(* CODESYS project Tc3_BAR_Common.library
   Company: Beckhoff
   Description: Library of implamentation common staff
   Version: 0.5.0
   DocFormat: reStructuredText
   Placeholder: Tc3_BAR_Common
   Author: Nikita Sakhnenko
   Title: Tc3_BAR_Common

Project tree, tasks and I/O mapping:
  libraries: Tc2_Standard, * (Beckhoff Automation GmbH); Tc2_System, * (Beckhoff Automation GmbH); Tc2_Utilities, * (Beckhoff Automation GmbH); VisuDialogs, * (System)
  Alarm/
    VisuElements/
      visualisation AlarmRecord_ActAlm_600
      visualisation AlarmRecord_History_600
      visualisation Current_Alarms_800x550
      visualisation Current_Alarms_dialog
      visualisation History_Of_Alarms_800x550
      visualisation History_Of_Alarms_dialog
    AlarmDiagram_1
    function block FB_Alarm [ST]: a1_Local_Quit, a2_Alarm_ScadaQuit, a3_Alarm_NoQuit, a4_Warning_RecordOnly, FB_init
    global variables LibAlarm
    program PRG_Alarms_Core [ST]: Blink, Current_Alarms_HMI, FB_Alarm_Execution, Get_Current_Time, History_Alarms_HMI
  Common/
    function TIME_TO_STRING_CE [ST]
    function TIME_TO_WSTRING_CE [ST]
    function TIME_TO_WSTRING_HMI [ST]
    function TS_to_STRING [ST]
    function TS_to_WSTRING [ST]
  DUTs/
    data type AlarmType
    data type E_AlarmColors
    data type ST_AlarmInfo
    data type ST_AlarmRecord
  InputVisu/
    visualisation TimeInput
  IO_terminals/
    DUTs/
      data type E_TermType
      data type TermChannel
    VisuElements/
      visualisation VisuAnalogChannel_Filled
      visualisation VisuAnalogChannel_Holow
    function block FB_AnalogChannel [ST]
  NC PTP Time Calculator/
    function block FB_7_SegTraj_Calculator [ST]: Step_1_Vmax_Amax_IsReachable, Step_2_Ta_Less_Than_Zero, Step_2_Td_Less_Than_Zero, Step_3_Gamma_Decrease_Seq
  Project Information/
    function F_GetCompany [ST]
    function F_GetTitle [ST]
    function F_GetVersion [ST]
  Trends/
    FBs/
      data type E_Trend_VISU_Type
      function block FB_TrendChanel [ST]: FB_init
      data type VisuStructPoint
    VISU/
      visualisation Trend_800_480
  Version/
    global variables Global_Version
  text list GlobalTextList
*)

// DUTs/AlarmType
{attribute 'qualified_only'}
{attribute 'strict'}
(*Вид аварийной блокировки*)
TYPE AlarmType :
(
	Alarm_LocalQuit 	:= 0,
	Alarm_ScadaQuit 	:= 1,
	Alarm_NoQuit 		:= 2,
	Warning_RecordOnly	:= 3,
	Warning_Type2		:= 4
);
END_TYPE

// DUTs/E_AlarmColors
{attribute 'qualified_only'}
{attribute 'strict'}
TYPE E_AlarmColors :
(
	E_Gray 		:= 16#7FD0D0D0, // Серый цвет
	E_Red  		:= 16#7FFF3C3C, // Красный цвет
	E_Yellow	:= 16#7FFFFF7D, // Желтый цвет
	E_green 	:= 16#7F00FF40, // Зеленый цвет
	E_Blue 		:= 16#7F8080FF  // Синий цвет
) DWORD;
END_TYPE

// DUTs/ST_AlarmInfo
(*Структура описания аварии*)
TYPE ST_AlarmInfo :
STRUCT
	AlarmID: WSTRING(5);				(*Текстовый идентификатор аварии*)
	Color: E_ALarmColors:=E_ALarmColors.E_Gray;		(*Цвет аварии. Заваисит от типа аварии*)
	Description: WSTRING(80):="--------------------------------------------------"; (*Поле описание аварии*)
	PossibleCause: WSTRING; 			(*Поле возможной причины аварии или указаний на аварийный узел*)
END_STRUCT
END_TYPE

// DUTs/ST_AlarmRecord
(*Структура записи в журнале аварий*)
TYPE ST_AlarmRecord EXTENDS ST_AlarmInfo :
STRUCT
	Time_On: 	WSTRING(20):="Нет данных"; 	(*Время возникновения аварии*)
	Time_Off: 	WSTRING(20):="Нет данных";	(*Время ухода аварии*)
	Time_Quit:	WSTRING(20):="Нет данных";	(*Время квитирования аварии*)
	isActive: BOOL;							(*Блокировка активна в настоящий момент*)
	wasQuited: BOOL;
END_STRUCT
END_TYPE

// IO_terminals/DUTs/E_TermType
{attribute 'qualified_only'}
{attribute 'strict'}
TYPE E_TermType :
(
	EL320x:=0,
	EL306x:=1,
	EL305x:=2,
	EL400x:=3,
	EL401x:=4,
	EL401x_4_20:=5
);
END_TYPE

// IO_terminals/DUTs/TermChannel
TYPE TermChannel :
STRUCT
	Status: WORD; (*бит XX.0 Underrange; бит ХХ.1 -Overrange; бит ХХ.6 - ERROR*)
	Value: INT;
END_STRUCT
END_TYPE

// Trends/FBs/E_Trend_VISU_Type
{attribute 'qualified_only'}
{attribute 'strict'}
TYPE E_Trend_VISU_Type :
(
	E_VISU_800_480 := 0,
	E_VISU_4_3 :=1
);
END_TYPE

// Trends/FBs/VisuStructPoint
TYPE VisuStructPoint :
STRUCT
	iX: INT;
	iY: INT;
END_STRUCT
END_TYPE

// Alarm/LibAlarm
{attribute 'qualified_only'}
VAR_GLOBAL CONSTANT
	MAX_ALARMS_NUM : UINT:=1000; (*Максимальное число аварий в программе*)
	MAX_HISTORY_NUM: UINT:=1000; (*Глубина Аварийного журнала*)
END_VAR

VAR_GLOBAL PERSISTENT
	HistoryAlarmsArray: ARRAY [1..MAX_ALARMS_NUM] OF ST_AlarmRecord; (*Массив с историей аварий*)
END_VAR

VAR_GLOBAL
	Blink: BOOL; // Мыргалка
	
	iNumberOfAlarms: UINT; 													//Количество экземпляров FB_Alarms
	FB_Alarm_Iterator: 	ARRAY [1..MAX_ALARMS_NUM] OF POINTER TO FB_alarm; 	//Итератор экземпляров FB_Alarm для исполнения
	ActiveAlarmsArray: 	ARRAY [1..MAX_ALARMS_NUM] OF ST_AlarmRecord; 		//Массив с текущими авариями
	
	Global_TimeStr: 		WSTRING(20);//	Метка текущего времени
	bRemoteQuitAllAlarms: 	BOOL;	 	// 	Переменная для удаленного квитирования аварии
	bLocalQuitAllAlarms AT %I*: BOOL;	//	Переменная для локального квитирования аварии
	bAlarmButtonBlink: 		BOOL;	 	// 	В настоящий момент есть активные не квитированные аварии требующие сброса
END_VAR

// Version/Global_Version
{attribute 'TcGenerated'}
{attribute 'no-analysis'}
{attribute 'linkalways'}
// This function has been automatically generated from the project information.
VAR_GLOBAL CONSTANT
	{attribute 'const_non_replaced'}
	stLibVersion_Tc3_BAR_Common : ST_LibVersion := (iMajor := 0, iMinor := 5, iBuild := 0, iRevision := 0, nFlags := 0, sVersion := '0.5.0');
END_VAR

// Alarm/FB_Alarm
{region "Documentation"}
(*
Функциональный блок обработки аварии
====================================
:Date: 2019-11-21
Служит для отображения аварий в текущем списке аварий и ведения истории.
В одном проекте может быть обьявлено максимум 1000 функциональных блоков FB_Alarm.
Максимальная глубина журнала аварий 1000.

Принцип использования
=====================
1. В библиотеке есть готовые экземпляры визуализации с таблицей текущих активных аварий: *Current_Alarms*
	и журналом аварий *History_Alarms*. Их следует добавить в проект, если есть необходимость в графическом отображении.
2. Перед обьявлением экземпляров обязательно следует добавить в исполняемый код программу *PRG_Alarms_Core();* 	 
	В этой подпрограмме происходят вызовы всех экземпляров FB_Alarm, а также всё необходимое для корректной работы системы вцелом.
3. После объявления *FB_Alarm*. Все что требуется для его использования это задать параметры и аварийное условие.

4. По переднему фронту *fbAlarm.AlarmEvent* активируется аварийная блокировка ("1" на выходе fbAlarm.isActive).
	 По заднему фронту входа *fbAlarm.AlarmEvent*Аварийная блокировкка снимется ("0" на выходе fbAlarm.isActive) в зависимости от типа аварии: 
====================  ========================================================
Alarm_Type           	Поведение по заднему фронту *fbAlarm.AlarmEvent*
====================  ========================================================
Local_Quit       		Снимается только после локального квитирования аварии
	 					LibAlarms.bLocalQuitAllAlarms - глобальная переменная 
						сброса квитирования всех активных аварий
						fbAlarm.bQuitAlarm - квитирование аварии экземпляра ФБ                 		
Alarm_ScadaQuit    		Снимается только после локального квитирования аварии
	 					LibAlarms.bLocalQuitAllAlarms - глобальная переменная 
						сброса квитирования всех активных аварий
	 					LibAlarms.bRemoteQuitAllAlarms - глобальная переменная 
						сброса квитирования всех активных аварий 							 
						fbAlarm.bQuitAlarm - квитирование аварии экземпляра ФБ
Alarm_NoQuit	    	Снимается сразу по заднему фронту *fbAlarm.AlarmEvent*
	 					Если не была квитирована, то об этом появиться запись в
						журнале
Warning_RecordOnly   	Делает запись в журнал по переднему фронту *fbAlarm.AlarmEvent*
    	 			 	Снимается без квитирования.
===================   ========================================================
5. Для отображения списка текущих аварий нужно использовать диалоговое окно TcSakhnenko.Current_Allarms_dialog
	 Для отображения журнала аварий нужно использовать диалоговое окно TcSakhnenko.History_Of_Allarms_dialog
*)
{endregion}
FUNCTION_BLOCK FINAL FB_Alarm	
VAR_INPUT
	AlarmCheckIsEnable: 		BOOL:=TRUE;		(*Проверка аварийного условия активна*)
	AlarmEvent: 				BOOL:=FALSE; 	(*Условие срабатывания аварии*)
	bQuitAlarm:    				BOOL:=FALSE;	(*Команда на квитирование аварии, 1-квитирование*)
	AlarmType: 					AlarmType; 		(*Тип квитирования аварии*)
	AlarmInfo: ST_AlarmInfo; 
	AlarmActivationDelay: 		TIME; 			(*Задержка на срабатывание аварии*)
END_VAR
VAR_OUTPUT
	isActive: BOOL; 		(*Аварийая блокировка активна*)
	WasQuited: BOOL;		(*Авария была квитирована*)
END_VAR
VAR
	tDelay : TON;
	TempAlarmRec: ST_AlarmRecord;
	AlarmNum: UINT; 			(*Порядковый номер аварии*)
	iState: UINT;(*Состояние аварии*)
	i: UINT;
	n: UINT;
END_VAR

IF AlarmCheckIsEnable THEN 
	CASE  AlarmType OF
		00:
			a1_Local_Quit();
		01:
			a2_Alarm_ScadaQuit();
		02:
			a3_Alarm_NoQuit();
		03:
			a4_Warning_RecordOnly();
	END_CASE
END_IF

ACTION a1_Local_Quit:
(*Обработчик Аварии, которую необходимо квитировать. Только локально.*)
TempAlarmRec.wasQuited:=WasQuited;
TempAlarmRec.isActive:=isActive;

CASE iState OF
	0:(*Инициализация*)
		isActive:=FALSE;
		WasQuited:=FALSE;
		TempAlarmRec.wasQuited:=FALSE;
		TempAlarmRec.Time_Quit:="Не квитирована";
		TempAlarmRec.AlarmID:=AlarmInfo.AlarmID;
		TempAlarmRec.Color:=AlarmInfo.Color;
		TempAlarmRec.Description:=AlarmInfo.Description;
		TempAlarmRec.PossibleCause:=AlarmInfo.PossibleCause;
 		iState:=10;

	10:(*Авария не активна. Ожидание активации аварии*)
		tDelay(IN:=AlarmEvent, PT:=AlarmActivationDelay);
			
		IF tDelay.Q THEN (*Возникновение первой аварии*)
			TempAlarmRec.PossibleCause:=AlarmInfo.PossibleCause;
			tDelay(IN:=FALSE);
			iState:=20;
		END_IF

		IF isActive THEN (*Авария не была квитирована и возникла еще раз*)
			TempAlarmRec.PossibleCause:=AlarmInfo.PossibleCause;
			tDelay(IN:=FALSE);
			iState:=30;
		END_IF
		
	20: (*Запись Времени Аварии*)
		TempAlarmRec.Time_On:=LibAlarm.Global_TimeStr;
		isActive:=TRUE;
		iState:= 30;
		
	30: (*Ожидание квитирования аварии и ее ухода*)
		IF (LibAlarm.bLocalQuitAllAlarms OR bQuitAlarm) THEN 
			TempAlarmRec.Time_Quit:=LibAlarm.Global_TimeStr;
			WasQuited:=TRUE;
			iState:=40;
		END_IF

		IF NOT AlarmEvent THEN
			IF NOT WasQuited THEN
				TempAlarmRec.Time_OFF:=LibAlarm.Global_TimeStr;
				iState:=31;
			END_IF;
		END_IF
	31:(*Авария ушла но не квитирована*)
			IF (LibAlarm.bLocalQuitAllAlarms OR bQuitAlarm) THEN
				TempAlarmRec.Time_Quit:=LibAlarm.Global_TimeStr;
				WasQuited:=TRUE;

				FOR i:=0 TO (LibAlarm.MAX_HISTORY_NUM - 2) DO
					n:=LibAlarm.MAX_HISTORY_NUM-i;
					LibAlarm.HistoryAlarmsArray[n]:=LibAlarm.HistoryAlarmsArray[n-1];
				END_FOR;

				LibAlarm.HistoryAlarmsArray[1]:=TempAlarmRec;
				iState:=00;
			END_IF
		
		IF AlarmEvent THEN //авария пришла снова
			TempAlarmRec.Time_Quit:="Не квитирована";

			FOR i:=0 TO (LibAlarm.MAX_HISTORY_NUM - 2) DO
				n:=LibAlarm.MAX_HISTORY_NUM-i;
				LibAlarm.HistoryAlarmsArray[n]:=LibAlarm.HistoryAlarmsArray[n-1];
			END_FOR;
		
			LibAlarm.HistoryAlarmsArray[1]:=TempAlarmRec;
			
			iState:=10;
		END_IF
		
		40:(*Авария ушла и квитирована*)
			IF NOT AlarmEvent THEN
			TempAlarmRec.Time_OFF:=LibAlarm.Global_TimeStr;

				FOR i:=0 TO (LibAlarm.MAX_HISTORY_NUM - 2) DO
					n:=LibAlarm.MAX_HISTORY_NUM-i;
					LibAlarm.HistoryAlarmsArray[n]:=LibAlarm.HistoryAlarmsArray[n-1];
				END_FOR;
		
				LibAlarm.HistoryAlarmsArray[1]:=TempAlarmRec;

				iState:=0;
			END_IF
		
END_CASE
END_ACTION

ACTION a2_Alarm_ScadaQuit:
(*Обработчик Аварии, которую необходимо квитировать. Локально и удаленно.*)
TempAlarmRec.wasQuited:=WasQuited;
TempAlarmRec.isActive:=isActive;

CASE iState OF
	0:(*Инициализация*)
		isActive:=FALSE;
		WasQuited:=FALSE;
		TempAlarmRec.Time_Quit:="Не квитирована";
		TempAlarmRec.AlarmID:=AlarmInfo.AlarmID;
		TempAlarmRec.Color:=AlarmInfo.Color;
		TempAlarmRec.Description:=AlarmInfo.Description;
		TempAlarmRec.PossibleCause:=AlarmInfo.PossibleCause;
 		iState:=10;

	10:(*Авария не активна. Ожидание активации аварии*)
		tDelay(IN:=AlarmEvent, PT:=AlarmActivationDelay);
			
		IF tDelay.Q THEN (*Возникновение первой аварии*)
			TempAlarmRec.PossibleCause:=AlarmInfo.PossibleCause;
			tDelay(IN:=FALSE);
			iState:=20;
		END_IF

		IF isActive THEN (*Авария не была квитирована и возникла еще раз*)
			TempAlarmRec.PossibleCause:=AlarmInfo.PossibleCause;
			tDelay(IN:=FALSE);
			iState:=30;
		END_IF
		
	20: (*Запись Времени Аварии*)
		TempAlarmRec.Time_On:=LibAlarm.Global_TimeStr;
		isActive:=TRUE;
		iState:= 30;
		
	30: (*Ожидание квитирования аварии и ее ухода*)
		IF (LibAlarm.bLocalQuitAllAlarms OR bQuitAlarm OR LibAlarm.bRemoteQuitAllAlarms) THEN 
			TempAlarmRec.Time_Quit:=LibAlarm.Global_TimeStr;
			WasQuited:=TRUE;
			iState:=40;
		END_IF

		IF NOT AlarmEvent THEN
			IF NOT WasQuited THEN
				TempAlarmRec.Time_OFF:=LibAlarm.Global_TimeStr;
				iState:=31;
			END_IF;
		END_IF
	31:(*Авария ушла но не квитирована*)
			IF (LibAlarm.bLocalQuitAllAlarms OR bQuitAlarm OR LibAlarm.bRemoteQuitAllAlarms) THEN
				TempAlarmRec.Time_Quit:=LibAlarm.Global_TimeStr;
				WasQuited:=TRUE;

				FOR i:=0 TO (LibAlarm.MAX_HISTORY_NUM - 2) DO
					n:=LibAlarm.MAX_HISTORY_NUM-i;
					LibAlarm.HistoryAlarmsArray[n]:=LibAlarm.HistoryAlarmsArray[n-1];
				END_FOR;

				LibAlarm.HistoryAlarmsArray[1]:=TempAlarmRec;
				iState:=00;
			END_IF

		IF AlarmEvent THEN
			TempAlarmRec.Time_Quit:="Не квитирована";

			FOR i:=0 TO (LibAlarm.MAX_HISTORY_NUM - 2) DO
				n:=LibAlarm.MAX_HISTORY_NUM-i;
				LibAlarm.HistoryAlarmsArray[n]:=LibAlarm.HistoryAlarmsArray[n-1];
			END_FOR;
		
			LibAlarm.HistoryAlarmsArray[1]:=TempAlarmRec;
			
			iState:=10;
		END_IF
		
		40:(*Авария ушла и квитирована*)
			IF NOT AlarmEvent THEN
			TempAlarmRec.Time_OFF:=LibAlarm.Global_TimeStr;

				FOR i:=0 TO (LibAlarm.MAX_HISTORY_NUM - 2) DO
					n:=LibAlarm.MAX_HISTORY_NUM-i;
					LibAlarm.HistoryAlarmsArray[n]:=LibAlarm.HistoryAlarmsArray[n-1];
				END_FOR;
		
				LibAlarm.HistoryAlarmsArray[1]:=TempAlarmRec;

				iState:=0;
			END_IF
		
END_CASE
END_ACTION

ACTION a3_Alarm_NoQuit:
(*Обработчик Аварии, которую необходимо квитировать*)
TempAlarmRec.wasQuited:=WasQuited;
TempAlarmRec.isActive:=isActive;

CASE iState OF
	0:(*Инициализация*)
		isActive:=FALSE;
		WasQuited:=FALSE;
		TempAlarmRec.Time_Quit:="Не квитирована";
		TempAlarmRec.AlarmID:=AlarmInfo.AlarmID;
		TempAlarmRec.Color:=AlarmInfo.Color;
		TempAlarmRec.Description:=AlarmInfo.Description;
		TempAlarmRec.PossibleCause:=AlarmInfo.PossibleCause;
 		iState:=10;

	10:(*Авария не активна. Ожидание активации аварии*)
		tDelay(IN:=AlarmEvent, PT:=AlarmActivationDelay);
			
		IF tDelay.Q THEN (*Возникновение первой аварии*)
			TempAlarmRec.PossibleCause:=AlarmInfo.PossibleCause;
			tDelay(IN:=FALSE);
			iState:=20;
		END_IF

		IF isActive THEN (*Авария не была квитирована и возникла еще раз*)
			TempAlarmRec.PossibleCause:=AlarmInfo.PossibleCause;
			tDelay(IN:=FALSE);
			iState:=30;
		END_IF
		
	20: (*Запись Времени Аварии*)
		TempAlarmRec.Time_On:=LibAlarm.Global_TimeStr;
		isActive:=TRUE;
		iState:= 30;
		
	30: (*Ожидание квитирования аварии и ее ухода*)
		IF (LibAlarm.bLocalQuitAllAlarms OR bQuitAlarm OR LibAlarm.bRemoteQuitAllAlarms) THEN 
			TempAlarmRec.Time_Quit:=LibAlarm.Global_TimeStr;
			WasQuited:=TRUE;
			iState:=40;
		END_IF

		IF NOT AlarmEvent THEN
			IF NOT WasQuited THEN
				TempAlarmRec.Time_OFF:=LibAlarm.Global_TimeStr;
				iState:=40;
			END_IF;
		END_IF
		
		40:(*Авария ушла и квитирована*)
			IF NOT AlarmEvent THEN
			TempAlarmRec.Time_OFF:=LibAlarm.Global_TimeStr;

				FOR i:=0 TO (LibAlarm.MAX_HISTORY_NUM - 2) DO
					n:=LibAlarm.MAX_HISTORY_NUM-i;
					LibAlarm.HistoryAlarmsArray[n]:=LibAlarm.HistoryAlarmsArray[n-1];
				END_FOR;
		
				LibAlarm.HistoryAlarmsArray[1]:=TempAlarmRec;

				iState:=0;
			END_IF
		
END_CASE
END_ACTION

ACTION a4_Warning_RecordOnly:
(*Предупреждение*)
CASE iState OF
	0:(*Инициализация*)
		isActive:=FALSE;
		WasQuited:=FALSE;
		TempAlarmRec.Time_Quit:="Не квитирована";
		TempAlarmRec.AlarmID:=AlarmInfo.AlarmID;
		TempAlarmRec.Color:=AlarmInfo.Color;
		TempAlarmRec.Description:=AlarmInfo.Description;
		TempAlarmRec.PossibleCause:=AlarmInfo.PossibleCause;
 		iState:=10;

	10:(*Авария не активна. Ожидание активации аварии*)
		tDelay(IN:=AlarmEvent, PT:=AlarmActivationDelay);
			
		IF tDelay.Q THEN (*Возникновение первой аварии*)
			tDelay(IN:=FALSE);
			
			TempAlarmRec.Time_ON:=LibAlarm.Global_TimeStr;
			TempAlarmRec.Time_Quit:="Не квитирована";
			TempAlarmRec.Time_OFF:=LibAlarm.Global_TimeStr;
			
				FOR i:=0 TO (LibAlarm.MAX_HISTORY_NUM - 2) DO
					n:=LibAlarm.MAX_HISTORY_NUM-i;
					LibAlarm.HistoryAlarmsArray[n]:=LibAlarm.HistoryAlarmsArray[n-1];
				END_FOR;
		
				LibAlarm.HistoryAlarmsArray[1]:=TempAlarmRec;
				
			iState:=20;
		END_IF

		
	20: (*Запись Времени Аварии*)
		IF NOT AlarmEvent THEN
			iState:=00;
		END_IF
		
END_CASE
END_ACTION

METHOD FB_init : BOOL
VAR_INPUT
	bInitRetains : BOOL; // if TRUE, the retain variables are initialized (warm start / cold start)
	bInCopyCode : BOOL;  // if TRUE, the instance afterwards gets moved into the copy code (online change)
END_VAR
libAlarm.iNumberOfAlarms:=libAlarm.iNumberOfAlarms+1;
AlarmNum:=libAlarm.iNumberOfAlarms;
LibAlarm.FB_Alarm_Iterator[AlarmNum]:=THIS;
END_METHOD

END_FUNCTION_BLOCK

// Alarm/PRG_Alarms_Core
PROGRAM PRG_Alarms_Core
VAR CONSTANT
	CurrentAlarmsDisplayNum: UINT:=10;//Количество отображаемых на экране текущих аварий
	HistoryAlarmsDisplayNum: UINT:=10;//Количество отображаемых на экране текущих аварий
END_VAR
VAR
	iFB: UINT; (*Итератор Функциональных блоков*)
	iCA: UINT; (*Итератор текущих аварий*)
	{region "Current_Alarms_HMI"}
	HMI_ActiveAlarms: ARRAY [1..CurrentAlarmsDisplayNum] OF ST_AlarmRecord;(*Масив с текущими отображаемыми авариями*)
	HMI_NumsAA : ARRAY[1..CurrentAlarmsDisplayNum] OF UINT;	(*Индексы в массиве текущих аварий*)
	iActiveAlarmsNumber: UINT;
	HMI_CurListAA: UINT;
	HMI_CurShiftAA: UINT;
	iHMI_AA: UINT;
	{endregion}
	
	{region "History_Alarms_HMI"}
	HMI_HistoryAlarms: ARRAY [1..HistoryAlarmsDisplayNum] OF ST_AlarmRecord;(*Масив с *)
	HMI_NumsHY : ARRAY[1..HistoryAlarmsDisplayNum] OF UINT;	(*Индексы в массиве истории аварий*)
	HMI_CurListHY: UINT;
	HMI_CurShiftHY: UINT;
	iHMI_HY: UINT;
	{endregion}
		 
	DefaultRec: ST_AlarmRecord;
	{region "Мыргалка"}
	t1: TON:=(PT:=T#1S);
	{endregion}
	
	{region "Get_Current_Time"}
	//Обновление строки текущего времени
	NT_GetTime: NT_GetTime;
	tonGetTime: TON:=(PT:=T#500MS);
	{endregion}
END_VAR

Get_Current_Time();

Blink();

FB_Alarm_Execution();

Current_Alarms_HMI();

History_Alarms_HMI();

ACTION Blink:
t1(in:=NOT t1.q);

IF t1.q THEN
LibAlarm.Blink:=NOT LibAlarm.Blink;
END_IF
END_ACTION

ACTION Current_Alarms_HMI:
	IF (HMI_CurShiftAA > LibAlarm.iNumberOfAlarms) THEN
		HMI_CurShiftAA:=LibAlarm.iNumberOfAlarms;
	ELSIF (HMI_CurShiftAA < 0 ) THEN
		HMI_CurShiftAA:=0;
	END_IF
	
	HMI_CurListAA := HMI_CurShiftAA / CurrentAlarmsDisplayNum;
	
	FOR iHMI_AA:=1 TO CurrentAlarmsDisplayNum DO
		HMI_NumsAA[iHMI_AA]:=iHMI_AA+HMI_CurShiftAA;
		HMI_ActiveAlarms[iHMI_AA]:=LibAlarm.ActiveAlarmsArray[HMI_NumsAA[iHMI_AA]];
	END_FOR
END_ACTION

ACTION FB_Alarm_Execution:
iCA:=1;
FOR iFB:=1 TO LibAlarm.iNumberOfAlarms DO
		LibAlarm.FB_Alarm_Iterator[iFB]^();
		LibAlarm.ActiveAlarmsArray[iFB]:=DefaultRec;
		IF LibAlarm.FB_Alarm_Iterator[iFB]^.isActive THEN
			LibAlarm.ActiveAlarmsArray[iCA]:=LibAlarm.FB_Alarm_Iterator[iFB]^.TempAlarmRec;
			iCA:=iCA+1;
		END_IF
END_FOR
END_ACTION

ACTION Get_Current_Time:
(*Получение текущего времени*)
tonGetTime(IN:= NOT tonGetTime.Q);
NT_GetTime(START:=tonGetTime.Q );
IF tonGetTime.Q THEN
	LibAlarm.Global_TimeStr := TS_to_WSTRING(NT_GetTime.TIMESTR);
END_IF
END_ACTION

ACTION History_Alarms_HMI:
	IF (HMI_CurShiftHY > (LibAlarm.MAX_HISTORY_NUM - HistoryAlarmsDisplayNum)) THEN
		HMI_CurShiftHY:=LibAlarm.MAX_HISTORY_NUM - HistoryAlarmsDisplayNum;
	ELSIF (HMI_CurShiftHY < 0 ) THEN
		HMI_CurShiftHY:=0;
	END_IF
	
	HMI_CurListHY := HMI_CurShiftHY / HistoryAlarmsDisplayNum;
	
	FOR iHMI_HY:=1 TO HistoryAlarmsDisplayNum DO
		HMI_NumsHY[iHMI_HY]:=iHMI_HY+HMI_CurShiftHY;
		HMI_HistoryAlarms[iHMI_HY]:=LibAlarm.HistoryAlarmsArray[HMI_NumsHY[iHMI_HY]];
	END_FOR
END_ACTION

END_PROGRAM

// Common/TS_to_WSTRING
FUNCTION TS_to_WSTRING : WSTRING(20)
VAR_INPUT
	in:TIMESTRUCT;
END_VAR
VAR
	str: WSTRING;
END_VAR

IF in.wHour>=10 THEN
str:=WCONCAT (str, WORD_TO_WSTRING(in.wHour));
ELSE
str:=WCONCAT (str, "0");
str:=WCONCAT (str, WORD_TO_WSTRING(in.wHour));
END_IF

str:=WCONCAT (str, ":");

IF in.wMinute>=10 THEN
str:=WCONCAT (str, WORD_TO_WSTRING(in.wMinute));
ELSE
str:=WCONCAT (str, "0");
str:=WCONCAT (str, WORD_TO_WSTRING(in.wMinute));
END_IF

str:=WCONCAT (str, ":");

IF in.wSecond>=10 THEN
str:=WCONCAT (str, WORD_TO_WSTRING(in.wSecond));
ELSE
str:=WCONCAT (str, "0");
str:=WCONCAT (str, WORD_TO_WSTRING(in.wSecond));
END_IF

str:=WCONCAT (str, " ");
str:=WCONCAT (str, WORD_TO_WSTRING(in.wDay));

IF in.wMonth <10 THEN
	str:=WCONCAT (str, ".0");
	str:=WCONCAT (str, WORD_TO_WSTRING(in.wMonth));	
ELSE
	str:=WCONCAT (str, ".");
	str:=WCONCAT (str, WORD_TO_WSTRING(in.wMonth));
END_IF

str:=WCONCAT (str, ".");
str:=WCONCAT (str, WORD_TO_WSTRING(in.wYear-2000));
TS_to_WSTRING:=str;

END_FUNCTION

// Common/TIME_TO_STRING_CE
FUNCTION TIME_TO_STRING_CE  : STRING(15)
VAR_INPUT
	InTime : TIME;
END_VAR
VAR
	DD: UINT;
	HH: UINT;
	MM: UINT;
	SS:UINT;
END_VAR

dd:=DWORD_TO_UINT (TIME_TO_DWORD(InTime) / TIME_TO_DWORD(T#1D));
HH:=DWORD_TO_UINT (TIME_TO_DWORD((InTime - T#24h*DD) / TIME_TO_DWORD(T#1h)));
MM:=DWORD_TO_UINT (TIME_TO_DWORD(InTime-T#24h*DD - T#60m*HH) / TIME_TO_DWORD(T#1m));
SS:=DWORD_TO_UINT (TIME_TO_DWORD(InTime - T#24h*DD - T#60m*HH - T#60s*MM) / TIME_TO_DWORD(T#1s));
TIME_TO_STRING_CE:=CONCAT(TIME_TO_STRING_CE, UINT_TO_STRING(DD));
TIME_TO_STRING_CE:=CONCAT(TIME_TO_STRING_CE, 'дн. ');
IF HH < 10 THEN
	TIME_TO_STRING_CE:=CONCAT(TIME_TO_STRING_CE, '0');
END_IF
TIME_TO_STRING_CE:=CONCAT(TIME_TO_STRING_CE, UINT_TO_STRING(HH));
TIME_TO_STRING_CE:=CONCAT(TIME_TO_STRING_CE, ':');
IF MM <10 THEN
	TIME_TO_STRING_CE:=CONCAT(TIME_TO_STRING_CE, '0');
END_IF
TIME_TO_STRING_CE:=CONCAT(TIME_TO_STRING_CE, UINT_TO_STRING(MM));
TIME_TO_STRING_CE:=CONCAT(TIME_TO_STRING_CE, ':');
IF SS <10 THEN
	TIME_TO_STRING_CE:=CONCAT(TIME_TO_STRING_CE, '0');
END_IF
TIME_TO_STRING_CE:=CONCAT(TIME_TO_STRING_CE, UINT_TO_STRING(SS));

END_FUNCTION

// Common/TIME_TO_WSTRING_CE
FUNCTION TIME_TO_WSTRING_CE  : WSTRING(15)
VAR_INPUT
	InTime : TIME;
END_VAR
VAR
	DD: UINT;
	HH: UINT;
	MM: UINT;
	SS:UINT;
END_VAR

dd:=DWORD_TO_UINT (TIME_TO_DWORD(InTime) / TIME_TO_DWORD(T#1D));
HH:=DWORD_TO_UINT (TIME_TO_DWORD((InTime - T#24h*DD) / TIME_TO_DWORD(T#1h)));
MM:=DWORD_TO_UINT (TIME_TO_DWORD(InTime-T#24h*DD - T#60m*HH) / TIME_TO_DWORD(T#1m));
SS:=DWORD_TO_UINT (TIME_TO_DWORD(InTime - T#24h*DD - T#60m*HH - T#60s*MM) / TIME_TO_DWORD(T#1s));
TIME_TO_WSTRING_CE:=WCONCAT(TIME_TO_WSTRING_CE, UINT_TO_WSTRING(DD));
TIME_TO_WSTRING_CE:=WCONCAT(TIME_TO_WSTRING_CE, "дн. ");
IF HH < 10 THEN
	TIME_TO_WSTRING_CE:=WCONCAT(TIME_TO_WSTRING_CE, "0");
END_IF
TIME_TO_STRING_CE:=WCONCAT(TIME_TO_WSTRING_CE, UINT_TO_WSTRING(HH));
TIME_TO_STRING_CE:=WCONCAT(TIME_TO_WSTRING_CE, ":");
IF MM <10 THEN
	TIME_TO_WSTRING_CE:=WCONCAT(TIME_TO_WSTRING_CE, "0");
END_IF
TIME_TO_WSTRING_CE:=WCONCAT(TIME_TO_WSTRING_CE, UINT_TO_WSTRING(MM));
TIME_TO_WSTRING_CE:=WCONCAT(TIME_TO_WSTRING_CE, ":");
IF SS <10 THEN
	TIME_TO_WSTRING_CE:=WCONCAT(TIME_TO_WSTRING_CE, "0");
END_IF
TIME_TO_WSTRING_CE:=WCONCAT(TIME_TO_WSTRING_CE, UINT_TO_WSTRING(SS));

END_FUNCTION

// Common/TIME_TO_WSTRING_HMI
FUNCTION TIME_TO_WSTRING_HMI  : WSTRING
VAR_INPUT
	InTime : TIME;
END_VAR
VAR
	DD: UINT;
	HH: UINT;
	MM: UINT;
	SS:UINT;
END_VAR

dd:=DWORD_TO_UINT (TIME_TO_DWORD(InTime) / TIME_TO_DWORD(T#1D));
HH:=DWORD_TO_UINT (TIME_TO_DWORD((InTime - T#24h*DD) / TIME_TO_DWORD(T#1h)));
MM:=DWORD_TO_UINT (TIME_TO_DWORD(InTime-T#24h*DD - T#60m*HH) / TIME_TO_DWORD(T#1m));
SS:=DWORD_TO_UINT (TIME_TO_DWORD(InTime - T#24h*DD - T#60m*HH - T#60s*MM) / TIME_TO_DWORD(T#1s));
IF (DD <> 00) THEN
	TIME_TO_WSTRING_HMI:=WCONCAT(TIME_TO_WSTRING_HMI, UINT_TO_WSTRING(DD));
	TIME_TO_WSTRING_HMI:=WCONCAT(TIME_TO_WSTRING_HMI, "дн. ");
END_IF
IF HH < 10 THEN
	TIME_TO_WSTRING_HMI:=WCONCAT(TIME_TO_WSTRING_HMI, "0");
END_IF
TIME_TO_WSTRING_HMI:=WCONCAT(TIME_TO_WSTRING_HMI, UINT_TO_WSTRING(HH));
TIME_TO_WSTRING_HMI:=WCONCAT(TIME_TO_WSTRING_HMI, ":");
IF MM <10 THEN
	TIME_TO_WSTRING_HMI:=WCONCAT(TIME_TO_WSTRING_HMI, "0");
END_IF
TIME_TO_WSTRING_HMI:=WCONCAT(TIME_TO_WSTRING_HMI, UINT_TO_WSTRING(MM));
TIME_TO_WSTRING_HMI:=WCONCAT(TIME_TO_WSTRING_HMI, ":");
IF SS <10 THEN
	TIME_TO_WSTRING_HMI:=WCONCAT(TIME_TO_WSTRING_HMI, "0");
END_IF
TIME_TO_WSTRING_HMI:=WCONCAT(TIME_TO_WSTRING_HMI, UINT_TO_WSTRING(SS));

END_FUNCTION

// Common/TS_to_STRING
FUNCTION TS_to_STRING : STRING(20)
VAR_INPUT
	in:TIMESTRUCT;
END_VAR
VAR
	str: STRING;
END_VAR

IF in.wHour>=10 THEN
str:=CONCAT (str, WORD_TO_STRING(in.wHour));
ELSE
str:=CONCAT (str, '0');
str:=CONCAT (str, WORD_TO_STRING(in.wHour));
END_IF

str:=CONCAT (str, ':');

IF in.wMinute>=10 THEN
str:=CONCAT (str, WORD_TO_STRING(in.wMinute));
ELSE
str:=CONCAT (str, '0');
str:=CONCAT (str, WORD_TO_STRING(in.wMinute));
END_IF

str:=CONCAT (str, ':');

IF in.wSecond>=10 THEN
str:=CONCAT (str, WORD_TO_STRING(in.wSecond));
ELSE
str:=CONCAT (str, '0');
str:=CONCAT (str, WORD_TO_STRING(in.wSecond));
END_IF

str:=CONCAT (str, ' ');
str:=CONCAT (str, WORD_TO_STRING(in.wDay));

IF in.wMonth <10 THEN
	str:=CONCAT (str, '.0');
	str:=CONCAT (str, WORD_TO_STRING(in.wMonth));	
ELSE
	str:=CONCAT (str, '.');
	str:=CONCAT (str, WORD_TO_STRING(in.wMonth));
END_IF

str:=CONCAT (str, '.');
str:=CONCAT (str, WORD_TO_STRING(in.wYear-2000));
TS_to_STRING:=str;

END_FUNCTION

// IO_terminals/FB_AnalogChannel
{region КОМЕНТЫ}
(**)

{endregion}
FUNCTION_BLOCK FINAL FB_AnalogChannel
VAR_INPUT
END_VAR
VAR_OUTPUT
	Underrange: BOOL; (*Недогрузка модульного канала*)
	Overrange: BOOL; (*Перегрузка модульного канала*)
	Error: BOOL; (*Ошибка модульного канала*)
END_VAR
VAR
	eTermType :E_TermType; (*Тип терминала ввода / вывода*)
	LowBound : LREAL; (*Нижняя граница диапазона изменения значений*)
	HighBound : LREAL:=100; (*Верхняя граница диапазона изменения значений*)
	Shift : LREAL; (*Значение сдвига диапазона изменения значений*)
	Value: LREAL; (*Текущее показание отмасштабированного канала*)
	
END_VAR
VAR_IN_OUT
	TerminalChannel : TermChannel; (*Ссылка на линкованный канал модуля*)
END_VAR

	CASE eTermType OF
		E_TermType.EL320x:
		
			Value:=INT_TO_LREAL(TerminalChannel.Value) * 0.1+Shift;
			
		E_TermType.EL306x:
			(*                  		  HighBound - LowBound                               *)
			(*  Value =lowbound +  ---------------------------------   x  ADC_Value + Shift;   *)
			(* 									32767   									  *)
			Value:= LowBound + ((HighBound - LowBound) * TerminalChannel.Value)/32676 + Shift;
			
		E_TermType.EL305x:
			(*                  		  HighBound - LowBound                               *)
			(*  Value =lowbound +  ---------------------------------   x  ADC_Value + Shift;   *)
			(* 									32767   									  *)
			Value:= LowBound + ((HighBound - LowBound) * TerminalChannel.Value)/32676 + Shift;
		
		E_TermType.EL400x:
			(*                           (Value-Lower_bound-Shift)*32767   		*)
			(*              ADC_Value = ------------------------------------    *)
			(*                              upper_bound-lower_bound          	*)
			TerminalChannel.Value:= LREAL_TO_INT( ((Value - LowBound - Shift)*32767)/(HighBound - LowBound));
			
		E_TermType.EL401x:
			(*                           (Value-Lower_bound-Shift)*32767   		*)
			(*              ADC_Value = ------------------------------------    *)
			(*                              upper_bound-lower_bound          	*)
			TerminalChannel.Value:= LREAL_TO_INT( ((Value - LowBound - Shift)*32767)/(HighBound - LowBound));
			
		E_TermType.EL401x_4_20:
			(*                (Value-Lower_bound-Shift)*(32767-6553) 	        *)
			(*  ADC_Value = ----------------------------------------  + 6553    *)
			(*                    upper_bound-lower_bound          	            *)
			TerminalChannel.Value:= LREAL_TO_INT( ((Value - LowBound - Shift)*(32767 -6553))/(HighBound - LowBound))+ 6553;	
	END_CASE
	
	Underrange:=TerminalChannel.Status.0;
	Overrange:=TerminalChannel.Status.1;
	Error:=TerminalChannel.Status.6;

END_FUNCTION_BLOCK

// NC PTP Time Calculator/FB_7_SegTraj_Calculator
//Расчет времен исполнения команд в NC PTP по семисегментной модели
// Написано на основе книги 
//
//	Trajectory Planning for Automatic Machines and Robots
//  Library of Congress Control Number: 2008934462
// 	Luigi Biagiotti · Claudio Melchiorri
//  Springer-Verlag Berlin Heidelberg 2008
//	ISBN: 978-3-540-85628-3   e-ISBN: 978-3-540-85629-0
//
//стр. 79 Параграф 3.4 Trajectory with Double S Velocity Profile
FUNCTION_BLOCK FB_7_SegTraj_Calculator
VAR_INPUT
	q_0, q_1 		: LREAL; 	// Начальная и конечная точки движния
	v_0, v_1 		: LREAL; 	// Начальное и конечное значения скорости
	v_max 			: LREAL:=1;	// Значение максимальной скорости
	a_max, a_min 	: LREAL:=1; // Максимальное и минимальное значения ускорения
	j_max, j_min 	: LREAL:=1; // Максимальное и минимальное значения рывка (производная от ускорения)
END_VAR
VAR_OUTPUT			
	T_j1, T_j2	: LREAL;// Время рывка ускорения и замедления 
	T_a		: LREAL; 	// Время ускорения
	T_d		: LREAL; 	// Время замедления скорения
	T_v		: LREAL; 	// Время постояной скорости
	T 		: LREAL; 	// Расчетное время 
	Error : BOOL; 		// Невозможно расчитать по введенным данным
END_VAR
VAR
	V_lim 			: LREAL; 	// Максимальновозможная скорость расчитаная на основе входных данных
	Delta 			: LREAL;
	Gamma			: LREAL:=1;
	Gamma_Shift 	: LREAL;
	A_max_lim 		: LREAL;
	
	A_lim_a 		: LREAL;
	A_lim_d 		: LREAL;
	
	Acc_MAX_CASE:   (A_max_IS_Reached,	A_max_IS_NOT_Reached);
	Acc_MIN_CASE:   (A_Min_IS_Reached,	A_Min_IS_NOT_Reached);

	i: UINT;
END_VAR

Error:=  a_max <> 0 AND v_max <> 0 AND j_max <> 0 AND v_max < v_0 ;

T_a:= T_d:= T_v:= T:= T_j1:= T_j2:= 0;

IF NOT Error THEN
	//Первая итерация расчета переменных. Предполагается что максимальная скорость и ускорение достижимы.
	Step_1_Vmax_Amax_IsReachable();	
	
	IF T_v > 0 THEN
		// Максимальная скорость и ускорение достижимы. Конец расчета
		T := T_a + T_v + T_d + 0.04;
		RETURN;
	ELSE
		// Максимальная скорость и ускорение не достижимы
		Gamma :=
		Gamma_Shift := 1;
		T_v := 0;
		Step_3_Gamma_Decrease_Seq();
		
		IF T_a < 0 OR T_d < 0 THEN
			Step_2_Ta_Less_Than_Zero();
			Step_2_Td_Less_Than_Zero();
			T := T_a + T_d + 0.04;
			RETURN;
		END_IF
		
		IF NOT (T_a > 2 * T_j1 AND T_d > 2 * T_j2) THEN
			FOR i:=1 TO 20 DO
				Step_3_Gamma_Decrease_Seq();
				Gamma_Shift := Gamma_Shift/2;
				IF NOT (T_a > 2 * T_j1 AND T_d > 2 * T_j2) THEN
					Gamma := Gamma - Gamma_Shift;
				ELSE
					Gamma := Gamma + Gamma_Shift;
				END_IF
				IF Gamma > 1 THEN
					Gamma := 1;
				END_IF
			END_FOR
		END_IF
		
		IF T_a < 0 OR T_d < 0 THEN
			Step_2_Ta_Less_Than_Zero();
			Step_2_Td_Less_Than_Zero();
			T := T_a + T_d + 0.04;
			RETURN;
		END_IF
		
		T := T_a + T_d+ 0.04;
	END_IF
END_IF

ACTION Step_1_Vmax_Amax_IsReachable:
IF (v_max - v_0) * j_max < a_max * a_max THEN
	Acc_MAX_CASE := A_max_IS_NOT_Reached;
ELSE
	Acc_MAX_CASE := A_max_IS_Reached;
END_IF

CASE Acc_MAX_CASE OF
	A_max_IS_NOT_Reached:
		T_j1:= SQRT((v_max - v_0)/j_max);
		T_a := 2 * T_j1;
		
	A_max_IS_Reached:
		T_j1:= a_max/j_max;
		T_a := T_j1 + (v_max - v_0)/a_max;
END_CASE

IF (v_max - v_1) * j_max < a_max * a_max THEN
	Acc_MIN_CASE := A_Min_IS_NOT_Reached;
ELSE
	Acc_MIN_CASE := A_Min_IS_Reached;
END_IF

CASE Acc_MIN_CASE OF
	A_Min_IS_NOT_Reached:
	IF v_max >= v_1 THEN
		T_j2:= SQRT((v_max - v_1)/j_max);
		T_d := 2 * T_j2;
	END_IF

		
	A_Min_IS_Reached:
	IF v_max >= v_1 THEN
		T_j2:= a_max/j_max;
		T_d := T_j2 + (v_max - v_1)/a_max;
	END_IF

END_CASE

T_v :=	(q_1 - q_0)/v_max - (T_a/2)*(1+ v_0/v_max) - (T_d/2)*(1 + v_1/v_max);
END_ACTION

ACTION Step_2_Ta_Less_Than_Zero:
IF T_a < 0 AND v_0 > v_1 THEN
	T_a := 0;
	T_d := 2*(q_1-q_0)/(v_1+v_0);
	T_j2:= (j_max*(q_1 - q_0) - SQRT(j_max*(j_max*(q_1-q_0)*(q_1-q_0) + (v_1+v_0)*(v_1+v_0)*(v_1-v_0))))/(j_max*(v_1+v_0));
	
	A_lim_d := - j_max * T_j2;
END_IF
END_ACTION

ACTION Step_2_Td_Less_Than_Zero:
IF T_d < 0 AND v_0 > v_1 THEN
	T_d := 0;
	T_a := 2*(q_1-q_0)/(v_1+v_0);
	T_j1:= (j_max*(q_1 - q_0) - SQRT(j_max*(j_max*(q_1-q_0)*(q_1-q_0) + (v_1+v_0)*(v_1+v_0)*(v_1-v_0))))/(j_max*(v_1+v_0));
	
	A_lim_a := j_max * T_j1;
END_IF
END_ACTION

ACTION Step_3_Gamma_Decrease_Seq:
T_j1 := T_j2 := a_max * Gamma / j_max;

Delta := EXPT(a_max * Gamma,4)/(j_max *j_max)
	   + 2*(v_0 * v_0 + v_1 * v_1)
	   + a_max * Gamma *(4 * (q_1 - q_0) - 2 *(a_max * Gamma/j_max)*(v_0 + v_1));
	   
IF Delta >=0 THEN
	T_a	:= (EXPT(a_max * Gamma,2)/j_max - 2*v_0 + SQRT(Delta))/(2 * a_max * Gamma);
	T_d := (EXPT(a_max * Gamma,2)/j_max - 2*v_1 + SQRT(Delta))/(2 * a_max * Gamma);
END_IF
END_ACTION

END_FUNCTION_BLOCK

// Project Information/F_GetCompany
// This function has been automatically generated from the project information.
{attribute 'signature_flag' := '1073741824'}
{attribute 'TcGenerated'}
{attribute 'no-analysis'}
FUNCTION F_GetCompany : WSTRING
VAR_INPUT
	
END_VAR

F_GetCompany := "Beckhoff";

END_FUNCTION

// Project Information/F_GetTitle
// This function has been automatically generated from the project information.
{attribute 'signature_flag' := '1073741824'}
{attribute 'TcGenerated'}
{attribute 'no-analysis'}
FUNCTION F_GetTitle : WSTRING
VAR_INPUT
	
END_VAR

F_GetTitle := "Tc3_BAR_Common";

END_FUNCTION

// Project Information/F_GetVersion
// This function has been automatically generated from the project information.
{attribute 'signature_flag' := '1073741824'}
{attribute 'TcGenerated'}
{attribute 'no-analysis'}
FUNCTION F_GetVersion : ST_LibVersion
VAR_INPUT
	
END_VAR

F_GetVersion.iMajor := 0;
F_GetVersion.iMinor := 5;
F_GetVersion.iBuild := 0;
F_GetVersion.iRevision := 0;

END_FUNCTION

// Trends/FBs/FB_TrendChanel
//Функциональный блок для хранения и обработки данных, отображающихся на визуализациях в папке Treands/VISU
FUNCTION_BLOCK FINAL FB_TrendChanel
VAR CONSTANT
	POINTS_NUMBER : UINT := 700; 		// Количество точек, из которых состоит график
END_VAR
VAR_INPUT 
	InputData		: REAL; 			// Вход данных для отображения на графике
	UpdatePeriod	: TIME:=T#100MS;	// Период обновления данных на графике
	MinimalValue	: REAL;				// Максимальное значение данных по оси Y
	MaximalValue	: REAL:=100;		// Максимальное значение данных по оси Y
	TrendType		: E_Trend_Visu_Type;// Тип графика
END_VAR
VAR_OUTPUT
	X_AxisNames 	: ARRAY [1..10] OF REAL;		// Текстовые метки для оси X
	Y_AxisNames 	: ARRAY [1..15] OF WSTRING(15);	// Текстовые метки для оси Y
END_VAR
VAR
	UpdateTime: TON;
	pPoints   : POINTER TO ARRAY[1..POINTS_NUMBER] OF VisuStructPoint;
	XY_points : ARRAY[1..POINTS_NUMBER] OF VisuStructPoint;
	i: UINT;
END_VAR

IF UpdatePeriod >= T#100MS THEN
	UpdateTime(IN:=NOT UpdateTime.Q , PT:= UpdatePeriod);
END_IF

pPoints := ADR(XY_points);

IF UpdateTime.Q THEN
	X_AxisNames[1]:= MinimalValue;
	X_AxisNames[7]:= MaximalValue;
	FOR i:=2 TO 6 DO
		X_AxisNames[i]:=MinimalValue + ((MaximalValue - MinimalValue)/6)*(i-1);
	END_FOR
	
	FOR i:=1 TO 15 DO
		Y_AxisNames[i]:=TIME_TO_WSTRING_HMI(UINT_TO_WORD(i) * UpdatePeriod * 70);
		Y_AxisNames[i]:=WCONCAT("-",Y_AxisNames[i]);
	END_FOR
	
	FOR i:=1 TO POINTS_NUMBER-1 DO
		XY_points[POINTS_NUMBER - i + 1].iY:=XY_points[POINTS_NUMBER-i].iY;
	END_FOR
	CASE TrendType OF 
		 0: XY_points[1].iY:=450-REAL_TO_INT((InputData - MinimalValue)*420/(MaximalValue - MinimalValue ));
		 1: (*Добавится в случае добавления нового экрана графика*)
	END_CASE

END_IF

METHOD FB_init : BOOL
VAR_INPUT
	bInitRetains 	: BOOL; // if TRUE, the retain variables are initialized (warm start / cold start)
	bInCopyCode 	: BOOL;  // if TRUE, the instance afterwards gets moved into the copy code (online change)
END_VAR
pPoints:=ADR(XY_points);

FOR i:=1 TO POINTS_NUMBER DO
	XY_points[i].iX:=UINT_TO_INT(70+i);
	XY_points[i].iY:=450;
END_FOR
END_METHOD

END_FUNCTION_BLOCK

// Alarm/VisuElements/AlarmRecord_ActAlm_600
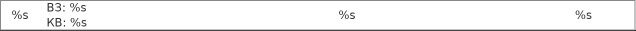
VISUALIZATION AlarmRecord_ActAlm_600  // 636x31
VAR_IN_OUT
	AlarmRecord: ST_AlarmRecord ; (*Запись об аварии для отображения*)
END_VAR
    Rectangle (163,0 368x30), "%s", text variable: AlarmRecord.Description, invisible if: (NOT AlarmRecord.isActive)
    Rectangle (40,0 123x15), "ВЗ: %s", text variable: AlarmRecord.Time_On, invisible if: (NOT AlarmRecord.isActive)
    Rectangle (40,15 123x15), "КВ: %s", text variable: AlarmRecord.Time_Quit, invisible if: (NOT AlarmRecord.isActive)
    Rectangle (0,0 40x30), "%s", text variable: AlarmRecord.AlarmID, invisible if: (NOT AlarmRecord.isActive)
    Rectangle (531,0 105x30), "%s", text variable: AlarmRecord.PossibleCause, invisible if: (NOT AlarmRecord.isActive)
    Line (0,30) (636,30), colour toggle: ((NOT AlarmRecord.wasQuited) AND LibAlarm.Blink), invisible if: (NOT AlarmRecord.isActive)
END_VISUALIZATION

// Alarm/VisuElements/AlarmRecord_History_600
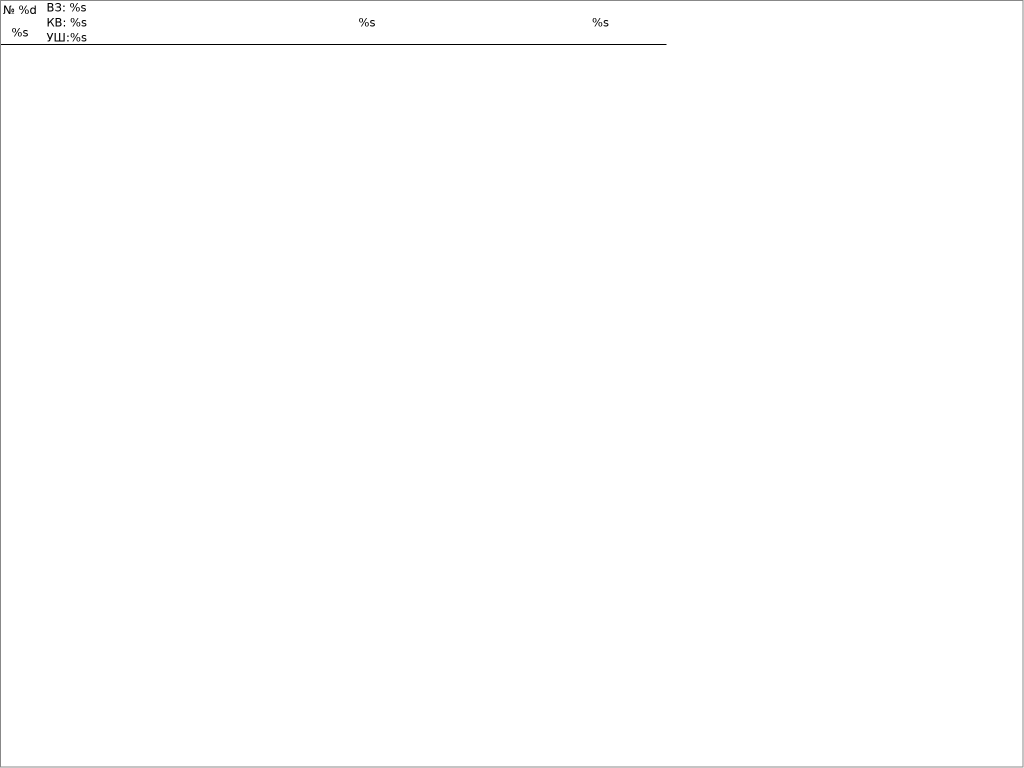
VISUALIZATION AlarmRecord_History_600  // 1024x768
VAR_IN_OUT
	AlarmRecord: ST_AlarmRecord ; (*Запись об аварии для отображения*)
	RecNum: UINT; (*Номер записи*)
END_VAR
    Rectangle (196,0 342x45), "%s", text variable: AlarmRecord.Description
    Rectangle (40,0 154x15), "ВЗ: %s", text variable: AlarmRecord.Time_On
    Rectangle (40,15 154x15), "КВ: %s", text variable: AlarmRecord.Time_Quit
    Rectangle (40,30 155x15), "УШ:%s", text variable: AlarmRecord.Time_Off
    Rectangle (538,0 125x45), "%s", text variable: AlarmRecord.PossibleCause
    Rectangle (0,20 40x25), "%s", text variable: AlarmRecord.AlarmID, colour variable: AlarmRecord.Color
    Rectangle (0,0 40x20), "№ %d", text variable: RecNum
    Line (0,44) (666,44)
END_VISUALIZATION

// Alarm/VisuElements/Current_Alarms_800x550
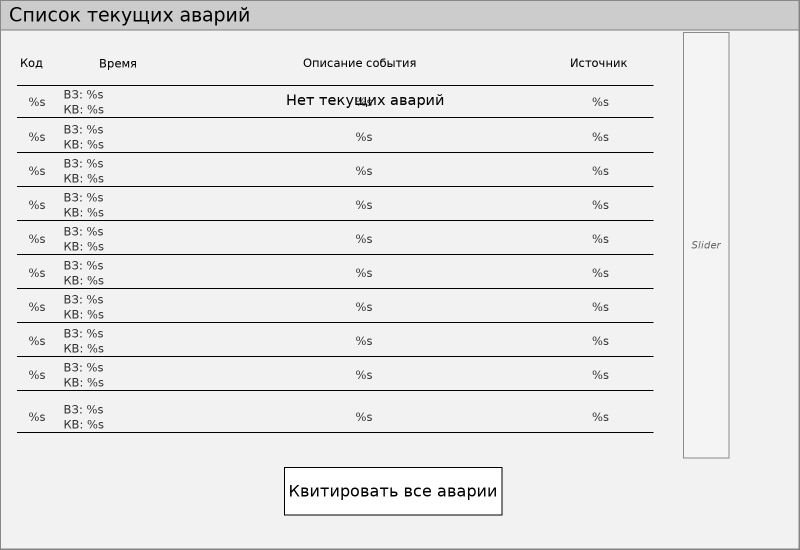
VISUALIZATION Current_Alarms_800x550  // 800x550
    Rectangle (0,0 800x550)
    Frame (17,122 600x30)
        shows AlarmRecord_ActAlm_600(AlarmRecord := PRG_Alarms_Core.HMI_ActiveAlarms[2])
    Frame (17,156 605x30)
        shows AlarmRecord_ActAlm_600(AlarmRecord := PRG_Alarms_Core.HMI_ActiveAlarms[3])
    Frame (17,190 605x30)
        shows AlarmRecord_ActAlm_600(AlarmRecord := PRG_Alarms_Core.HMI_ActiveAlarms[4])
    Frame (17,224 605x30)
        shows AlarmRecord_ActAlm_600(AlarmRecord := PRG_Alarms_Core.HMI_ActiveAlarms[5])
    Frame (17,258 605x30)
        shows AlarmRecord_ActAlm_600(AlarmRecord := PRG_Alarms_Core.HMI_ActiveAlarms[6])
    Frame (17,292 635x30)
        shows AlarmRecord_ActAlm_600(AlarmRecord := PRG_Alarms_Core.HMI_ActiveAlarms[7])
    Frame (17,326 635x30)
        shows AlarmRecord_ActAlm_600(AlarmRecord := PRG_Alarms_Core.HMI_ActiveAlarms[8])
    Frame (17,360 635x30)
        shows AlarmRecord_ActAlm_600(AlarmRecord := PRG_Alarms_Core.HMI_ActiveAlarms[9])
    Frame (17,402 639x32)
        shows AlarmRecord_ActAlm_600(AlarmRecord := PRG_Alarms_Core.HMI_ActiveAlarms[10])
    Label (250,85 231x30), "Нет текущих аварий", invisible if: PRG_Alarms_Core.HMI_ActiveAlarms[1].isActive
    Frame (17,87 641x31)
        shows AlarmRecord_ActAlm_600(AlarmRecord := PRG_Alarms_Core.HMI_ActiveAlarms[1])
    Rectangle (0,0 800x30), "Список текущих аварий"
    Slider (683,32 46x426), variable: PRG_Alarms_Core.HMI_CurShiftAA, scale 0..1000
    Label (17,48 37x30), "Код"
    Label (300,48 216x30), "Описание события"
    Label (567,48 77x30), "Источник"
    Label (92,54 52x19), "Время"
    Line (17,85) (653,85)
    RoundedRectangle (284,467 218x48), "Квитировать все аварии"
        tap LibAlarm.bLocalQuitAllAlarms
END_VISUALIZATION

// Alarm/VisuElements/Current_Alarms_dialog
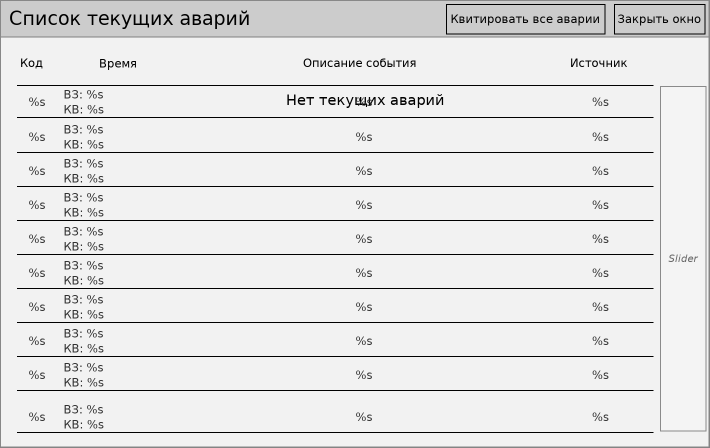
VISUALIZATION Current_Alarms_dialog  // 710x448
    Rectangle (0,0 710x448)
    Frame (17,122 600x30)
        shows AlarmRecord_ActAlm_600(AlarmRecord := PRG_Alarms_Core.HMI_ActiveAlarms[2])
    Frame (17,156 605x30)
        shows AlarmRecord_ActAlm_600(AlarmRecord := PRG_Alarms_Core.HMI_ActiveAlarms[3])
    Frame (17,190 605x30)
        shows AlarmRecord_ActAlm_600(AlarmRecord := PRG_Alarms_Core.HMI_ActiveAlarms[4])
    Frame (17,224 605x30)
        shows AlarmRecord_ActAlm_600(AlarmRecord := PRG_Alarms_Core.HMI_ActiveAlarms[5])
    Frame (17,258 605x30)
        shows AlarmRecord_ActAlm_600(AlarmRecord := PRG_Alarms_Core.HMI_ActiveAlarms[6])
    Frame (17,292 635x30)
        shows AlarmRecord_ActAlm_600(AlarmRecord := PRG_Alarms_Core.HMI_ActiveAlarms[7])
    Frame (17,326 635x30)
        shows AlarmRecord_ActAlm_600(AlarmRecord := PRG_Alarms_Core.HMI_ActiveAlarms[8])
    Frame (17,360 635x30)
        shows AlarmRecord_ActAlm_600(AlarmRecord := PRG_Alarms_Core.HMI_ActiveAlarms[9])
    Frame (17,402 639x32)
        shows AlarmRecord_ActAlm_600(AlarmRecord := PRG_Alarms_Core.HMI_ActiveAlarms[10])
    Label (250,85 231x30), "Нет текущих аварий", invisible if: PRG_Alarms_Core.HMI_ActiveAlarms[1].isActive
    Frame (17,87 641x31)
        shows AlarmRecord_ActAlm_600(AlarmRecord := PRG_Alarms_Core.HMI_ActiveAlarms[1])
    Rectangle (0,0 710x37), "Список текущих аварий"
    Slider (660,86 46x345), variable: PRG_Alarms_Core.HMI_CurShiftAA, scale 0..1000
    Label (17,48 37x30), "Код"
    Label (300,48 216x30), "Описание события"
    Label (567,48 77x30), "Источник"
    Label (92,54 52x19), "Время"
    Line (17,85) (653,85)
    RoundedRectangle (614,4 91x30), "Закрыть окно"
        OnMouseClick:  Dialog=Current_Alarms_dialog, Result=OK, NumpadKeypadSet=True
    RoundedRectangle (446,4 159x30), "Квитировать все аварии"
        tap LibAlarm.bLocalQuitAllAlarms
END_VISUALIZATION

// Alarm/VisuElements/History_Of_Alarms_800x550
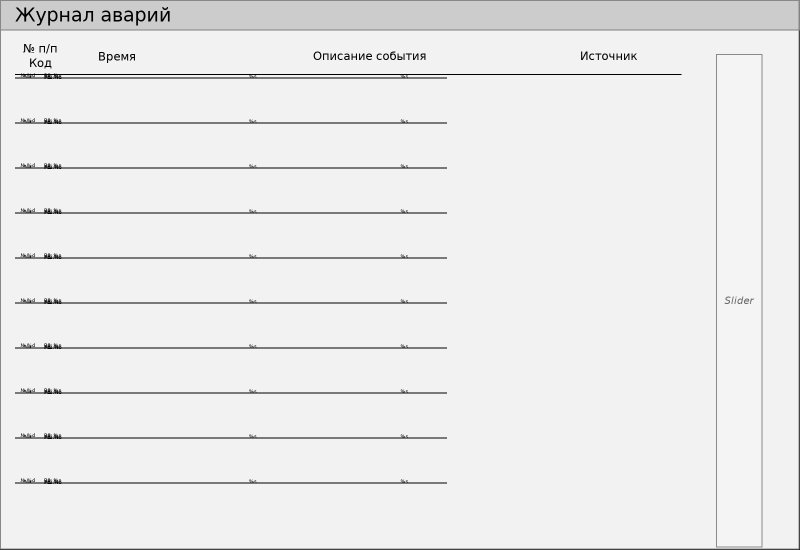
VISUALIZATION History_Of_Alarms_800x550  // 800x550
    Rectangle (0,0 800x550)
    Frame (15,75 664x46)
        shows AlarmRecord_History_600(AlarmRecord := PRG_Alarms_Core.HMI_HistoryAlarms[1], RecNum := PRG_Alarms_Core.HMI_NumsHY[1])
    Frame (15,120 664x46)
        shows AlarmRecord_History_600(AlarmRecord := PRG_Alarms_Core.HMI_HistoryAlarms[2], RecNum := PRG_Alarms_Core.HMI_NumsHY[2])
    Frame (15,165 664x46)
        shows AlarmRecord_History_600(AlarmRecord := PRG_Alarms_Core.HMI_HistoryAlarms[3], RecNum := PRG_Alarms_Core.HMI_NumsHY[3])
    Frame (15,210 664x46)
        shows AlarmRecord_History_600(AlarmRecord := PRG_Alarms_Core.HMI_HistoryAlarms[4], RecNum := PRG_Alarms_Core.HMI_NumsHY[4])
    Frame (15,255 664x46)
        shows AlarmRecord_History_600(AlarmRecord := PRG_Alarms_Core.HMI_HistoryAlarms[5], RecNum := PRG_Alarms_Core.HMI_NumsHY[5])
    Frame (15,300 664x46)
        shows AlarmRecord_History_600(AlarmRecord := PRG_Alarms_Core.HMI_HistoryAlarms[6], RecNum := PRG_Alarms_Core.HMI_NumsHY[6])
    Frame (15,345 664x46)
        shows AlarmRecord_History_600(AlarmRecord := PRG_Alarms_Core.HMI_HistoryAlarms[7], RecNum := PRG_Alarms_Core.HMI_NumsHY[7])
    Frame (15,390 664x46)
        shows AlarmRecord_History_600(AlarmRecord := PRG_Alarms_Core.HMI_HistoryAlarms[8], RecNum := PRG_Alarms_Core.HMI_NumsHY[8])
    Frame (15,435 664x46)
        shows AlarmRecord_History_600(AlarmRecord := PRG_Alarms_Core.HMI_HistoryAlarms[9], RecNum := PRG_Alarms_Core.HMI_NumsHY[9])
    Frame (15,480 664x46)
        shows AlarmRecord_History_600(AlarmRecord := PRG_Alarms_Core.HMI_HistoryAlarms[10], RecNum := PRG_Alarms_Core.HMI_NumsHY[10])
    Slider (716,54 46x493), variable: PRG_Alarms_Core.HMI_CurShiftHY, scale 0..1000
    Label (17,41 47x30), "№ п/п Код"
    Label (310,41 216x30), "Описание события"
    Label (577,41 77x30), "Источник"
    Label (91,47 52x19), "Время"
    Line (15,74) (681,74)
    Rectangle (0,0 800x30), "Журнал аварий"
END_VISUALIZATION

// Alarm/VisuElements/History_Of_Alarms_dialog
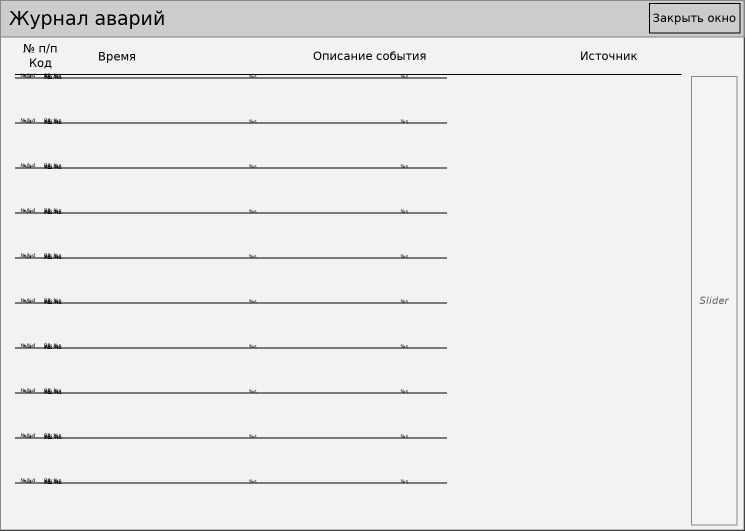
VISUALIZATION History_Of_Alarms_dialog  // 745x531
    Rectangle (0,0 745x531)
    Frame (15,75 664x46)
        shows AlarmRecord_History_600(AlarmRecord := PRG_Alarms_Core.HMI_HistoryAlarms[1], RecNum := PRG_Alarms_Core.HMI_NumsHY[1])
    Frame (15,120 664x46)
        shows AlarmRecord_History_600(AlarmRecord := PRG_Alarms_Core.HMI_HistoryAlarms[2], RecNum := PRG_Alarms_Core.HMI_NumsHY[2])
    Frame (15,165 664x46)
        shows AlarmRecord_History_600(AlarmRecord := PRG_Alarms_Core.HMI_HistoryAlarms[3], RecNum := PRG_Alarms_Core.HMI_NumsHY[3])
    Frame (15,210 664x46)
        shows AlarmRecord_History_600(AlarmRecord := PRG_Alarms_Core.HMI_HistoryAlarms[4], RecNum := PRG_Alarms_Core.HMI_NumsHY[4])
    Frame (15,255 664x46)
        shows AlarmRecord_History_600(AlarmRecord := PRG_Alarms_Core.HMI_HistoryAlarms[5], RecNum := PRG_Alarms_Core.HMI_NumsHY[5])
    Frame (15,300 664x46)
        shows AlarmRecord_History_600(AlarmRecord := PRG_Alarms_Core.HMI_HistoryAlarms[6], RecNum := PRG_Alarms_Core.HMI_NumsHY[6])
    Frame (15,345 664x46)
        shows AlarmRecord_History_600(AlarmRecord := PRG_Alarms_Core.HMI_HistoryAlarms[7], RecNum := PRG_Alarms_Core.HMI_NumsHY[7])
    Frame (15,390 664x46)
        shows AlarmRecord_History_600(AlarmRecord := PRG_Alarms_Core.HMI_HistoryAlarms[8], RecNum := PRG_Alarms_Core.HMI_NumsHY[8])
    Frame (15,435 664x46)
        shows AlarmRecord_History_600(AlarmRecord := PRG_Alarms_Core.HMI_HistoryAlarms[9], RecNum := PRG_Alarms_Core.HMI_NumsHY[9])
    Frame (15,480 664x46)
        shows AlarmRecord_History_600(AlarmRecord := PRG_Alarms_Core.HMI_HistoryAlarms[10], RecNum := PRG_Alarms_Core.HMI_NumsHY[10])
    Slider (691,76 46x449), variable: PRG_Alarms_Core.HMI_CurShiftHY, scale 0..1000
    Label (17,41 47x30), "№ п/п Код"
    Label (310,41 216x30), "Описание события"
    Label (577,41 77x30), "Источник"
    Label (91,47 52x19), "Время"
    Line (15,74) (681,74)
    Rectangle (0,0 745x37), "Журнал аварий"
    RoundedRectangle (649,3 91x30), "Закрыть окно"
        OnMouseClick:  Dialog=History_Of_Alarms_dialog, Result=OK, NumpadKeypadSet=True
END_VISUALIZATION

// InputVisu/TimeInput
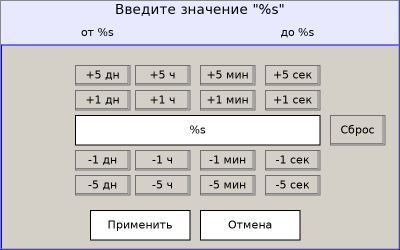
VISUALIZATION TimeInput  // 400x250
VAR_INPUT
	stVariableValue : STRING;
	stMin : STRING;
	stMax : STRING;
	wstTitle : WSTRING;
	flags : DWORD;
END_VAR
VAR
	bInit 			: BOOL;
	stMessage 		: STRING;
	stOutputValue 	: STRING;
	iCaretPosition	: INT;
	iSelectionStart	: INT;
	iSelectionEnd	: INT;
	xAllSelected	: BOOL;
END_VAR
    Rectangle (0,0 400x250)
    Rectangle (200,210 100x30), "Отмена"
        OnMouseDown:  Dialog=TimeInput, Result=Cancel, NumpadKeypadSet=True
    Rectangle (90,210 100x30), "Применить"
        OnMouseUp:  Dialog=TimeInput, Result=Yes, NumpadKeypad=True, NumpadKeypadSet=True
    Rectangle (0,0 400x45), "Введите значение "%s"", text variable: Header
    Button (265,90 55x20), "+1 сек", invisible if: (MinTime + T#1s >= MaxTime)
        OnMouseUp: execute {
            IF ((timevar+T#1S <= MaxTime ) AND
            			(timevar+T#1S > TimeVar)) THEN
            	timevar:=timevar+T#1S;
            END_IF
        }
    Rectangle (75,115 245x30), "%s", text variable: TIME_TO_WSTRING_HMI(TimeVar)
        p4168582468: "Время"
    Button (265,65 55x20), "+5 сек", invisible if: (MinTime + T#5s >= MaxTime)
        OnMouseUp: execute {
            IF ((timevar+T#5S <= MaxTime ) AND
            			(timevar+T#5S > TimeVar)) THEN
            	timevar:=timevar+T#5S;
            ELSE
            	timevar:=MaxTime;
            END_IF
        }
    Button (265,175 55x20), "-5 сек", invisible if: (MinTime + T#5s) >= MaxTime
        OnMouseUp: execute {
            IF (((timevar-T#5S) >= MinTime)AND
            				(timevar-T#5S < timevar)) THEN
            	timevar:=timevar-T#5S;
            ELSE
            	TimeVar:=MinTime;
            END_IF
        }
    Button (265,150 55x20), "-1 сек", invisible if: (MinTime + T#1s) >= MaxTime
        OnMouseUp: execute {
            IF (((timevar-T#1S) >= MinTime)AND
            				(timevar-T#1S < timevar)) THEN
            	timevar:=timevar-T#1S;
            END_IF
        }
    Button (200,90 55x20), "+1 мин", invisible if: (MinTime + T#1m >= MaxTime)
        OnMouseUp: execute {
            IF ((timevar+T#1M <= MaxTime ) AND
            			(timevar+T#1M > TimeVar)) THEN
            	timevar:=timevar+T#1m;
            END_IF
        }
    Button (200,65 55x20), "+5 мин", invisible if: (MinTime + T#5m > MaxTime)
        OnMouseUp: execute {
            IF ((timevar+T#5M <= MaxTime ) AND
            			(timevar+T#5M > TimeVar)) THEN
            	timevar:=timevar+T#5M;
            ELSE
            	timevar:=MaxTime;
            END_IF
        }
    Button (135,90 55x20), "+1 ч", invisible if: (MinTime + T#1h >= MaxTime)
        OnMouseUp: execute {
            IF ((timevar+T#1H <= MaxTime ) AND
            			(timevar+T#1H > TimeVar)) THEN
            	timevar:=timevar+T#1H;
            END_IF
        }
    Button (135,65 55x20), "+5 ч", invisible if: (MinTime + T#5h >= MaxTime)
        OnMouseUp: execute {
            IF ((timevar+T#5H <= MaxTime ) AND
            			(timevar+T#5H > TimeVar)) THEN
            	timevar:=timevar+T#5h;
            ELSE
            	timevar:=MaxTime;
            END_IF
        }
    Button (200,175 55x20), "-5 мин", invisible if: (MinTime + T#5m) >= MaxTime
        OnMouseUp: execute {
            IF (((timevar-T#5M) >= MinTime)AND
            				(timevar-T#5M < timevar)) THEN
            	timevar:=timevar-T#5m;
            ELSE
            	TimeVar:=MinTime;
            END_IF
        }
    Button (200,150 55x20), "-1 мин", invisible if: (MinTime + T#1m) >=MaxTime
        OnMouseUp: execute {
            IF (((timevar-T#1M) >= MinTime)AND
            				(timevar-T#1M < timevar)) THEN
            	timevar:=timevar-T#1m;
            END_IF
        }
    Button (135,175 55x20), "-5 ч", invisible if: (MinTime + T#5h) >= MaxTime
        OnMouseUp: execute {
            IF (((timevar-T#5H) >= MinTime)AND
            				(timevar-T#5h < timevar)) THEN
            	timevar:=timevar-T#5H;
            ELSE
            	TimeVar:=MinTime;
            END_IF
        }
    Button (135,150 55x20), "-1 ч", invisible if: (MinTime + T#1h) >= MaxTime
        OnMouseUp: execute {
            IF (((timevar-T#1H) >= MinTime)AND
            				(timevar-T#1H < timevar)) THEN
            	timevar:=timevar-T#1h;
            END_IF
        }
    Button (75,90 55x20), "+1 дн", invisible if: (MinTime + T#1d >=MaxTime)
        OnMouseUp: execute {
            IF ((timevar+T#1D <= MaxTime ) AND
            			(timevar+T#1D > TimeVar)) THEN
            	timevar:=timevar+T#1d;
            END_IF
        }
    Button (75,65 55x20), "+5 дн", invisible if: (MinTime + T#5d >= MaxTime)
        OnMouseUp: execute {
            IF ((timevar+T#5D <= MaxTime ) AND
            			(timevar+T#5D > TimeVar)) THEN
            	timevar:=timevar+T#5D;
            ELSE
            	timevar:=MaxTime;
            END_IF
        }
    Button (75,175 55x20), "-5 дн", invisible if: (MinTime + T#5d) >= MaxTime
        OnMouseUp: execute {
            IF (((timevar-T#5D) >= MinTime)AND
            				(timevar-T#5D < timevar)) THEN
            	timevar:=timevar-T#5D;
            ELSE
            	TimeVar:=MinTime;
            END_IF
        }
    Button (75,150 55x20), "-1 дн", invisible if: (MinTime + T#1d) >= MaxTime
        OnMouseUp: execute {
            IF (((timevar-T#1D) >= MinTime)AND
            				(timevar-T#1D < timevar)) THEN
            	timevar:=timevar-T#1D;
            END_IF
        }
    Button (330,115 55x30), "Сброс"
        OnMouseUp: execute { timevar:=MinTime; }
    Rectangle (0,20 195x25), "от %s", text variable: TIME_TO_WSTRING_HMI(MinTime)
        p4168582468: "Время"
    Rectangle (195,20 205x25), "до %s", text variable: TIME_TO_WSTRING_HMI(MaxTime)
        p4168582468: "Время"
    hotkey  Id=481037385728, Key=KeyDown=True, KeyName=ESCAPE, VisuElemId=10
END_VISUALIZATION

// IO_terminals/VisuElements/VisuAnalogChannel_Filled
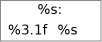
VISUALIZATION VisuAnalogChannel_Filled  // 102x42
VAR_INPUT
	Name: WSTRING;
	Unit: WSTRING;
END_VAR
VAR_IN_OUT
	fbAnalChan : FB_AnalogChannel;
END_VAR
    Rectangle (0,0 100x40), "%s:", text variable: Name, colour toggle: fbAnalChan.Error AND Tc3Sakhnenko.LibAlarm.Blink
        OnMouseDown: write fbAnalChan.Shift via Default, min 0, max 100
    Rectangle (0,20 55x20), "%3.1f", text variable: fbAnalChan.Value
    Rectangle (50,20 50x20), "%s", text variable: Unit
END_VISUALIZATION

// IO_terminals/VisuElements/VisuAnalogChannel_Holow
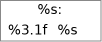
VISUALIZATION VisuAnalogChannel_Holow  // 102x42
VAR_INPUT
	Name: WSTRING;
	Unit: WSTRING;
END_VAR
VAR_IN_OUT
	fbAnalChan : FB_AnalogChannel;
END_VAR
    Rectangle (0,0 100x40), "%s:", text variable: Name, colour toggle: fbAnalChan.Error AND Tc3Sakhnenko.LibAlarm.Blink
        OnMouseDown: write fbAnalChan.Shift via Default, min 0, max 100
    Rectangle (0,20 55x20), "%3.1f", text variable: fbAnalChan.Value
    Rectangle (50,20 50x20), "%s", text variable: Unit
END_VISUALIZATION

// Trends/VISU/Trend_800_480
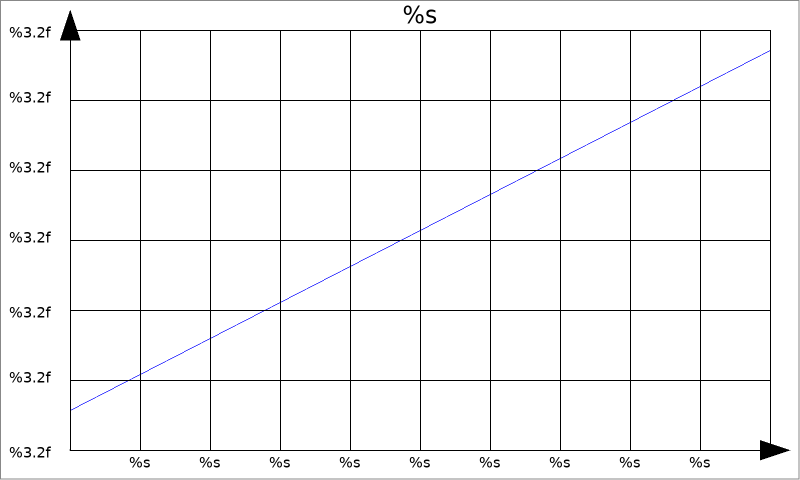
VISUALIZATION Trend_800_480  // 800x480
VAR_INPUT
	Header : WSTRING;
END_VAR
VAR_IN_OUT
	fb_TrendChanel1: FB_TrendChanel;
END_VAR
    Polyline (70,410) (770,50)
        p1285906596: fb_TrendChanel1.pPoints
        p3184209983: fb_TrendChanel1.POINTS_NUMBER
    Polygon (70,10) (80,40) (60,40)
    Line (70,380) (770,380)
    Line (70,310) (770,310)
    Line (70,240) (770,240)
    Line (70,170) (770,170)
    Line (70,100) (770,100)
    Rectangle (0,440 60x25), "%3.2f", text variable: fb_TrendChanel1.X_AxisNames[1]
    Rectangle (0,365 60x25), "%3.2f", text variable: fb_TrendChanel1.X_AxisNames[2]
    Rectangle (0,300 60x25), "%3.2f", text variable: fb_TrendChanel1.X_AxisNames[3]
    Rectangle (0,225 60x25), "%3.2f", text variable: fb_TrendChanel1.X_AxisNames[4]
    Rectangle (0,155 60x25), "%3.2f", text variable: fb_TrendChanel1.X_AxisNames[5]
    Rectangle (0,85 60x25), "%3.2f", text variable: fb_TrendChanel1.X_AxisNames[6]
    Rectangle (0,20 60x25), "%3.2f", text variable: fb_TrendChanel1.X_AxisNames[7]
    Rectangle (105,450 70x25), "%s", text variable: fb_TrendChanel1.Y_AxisNames[1]
    Rectangle (175,450 70x25), "%s", text variable: fb_TrendChanel1.Y_AxisNames[2]
    Rectangle (245,450 70x25), "%s", text variable: fb_TrendChanel1.Y_AxisNames[3]
    Rectangle (315,450 70x25), "%s", text variable: fb_TrendChanel1.Y_AxisNames[4]
    Rectangle (385,450 70x25), "%s", text variable: fb_TrendChanel1.Y_AxisNames[5]
    Rectangle (455,450 70x25), "%s", text variable: fb_TrendChanel1.Y_AxisNames[6]
    Rectangle (525,450 70x25), "%s", text variable: fb_TrendChanel1.Y_AxisNames[7]
    Rectangle (595,450 70x25), "%s", text variable: fb_TrendChanel1.Y_AxisNames[8]
    Rectangle (665,450 70x25), "%s", text variable: fb_TrendChanel1.Y_AxisNames[9]
    Rectangle (210,0 420x30), "%s", text variable: Header
    Line (70,30) (770,30)
    Line (140,30) (140,450)
    Line (210,30) (210,450)
    Line (280,30) (280,450)
    Line (350,30) (350,450)
    Line (420,30) (420,450)
    Line (490,30) (490,450)
    Line (560,30) (560,450)
    Line (630,30) (630,450)
    Line (700,30) (700,450)
    Polyline (70,20) (70,450) (770,450)
    Line (770,30) (770,450)
    Polygon (790,450) (760,460) (760,440)
END_VISUALIZATION
